ABB RAPID module: Data.modx

MODULE Data
     ! Home
    CONST robtarget rHomePos:=[[368.56,0,469.95],[0.0562068,-0.220361,0.97346,-0.0256232],[0,-1,-1,0],[9E+09,9E+09,9E+09,9E+09,9E+09,9E+09]];

    ! DipSchoko
    CONST robtarget rApprochPickBiscuit:=[[599.81,297.31,218.70],[0.0160586,-0.550955,-0.834314,-0.010557],[0,0,1,0],[9E+09,9E+09,9E+09,9E+09,9E+09,9E+09]];
    CONST robtarget rPickBiscuit:=[[446.88,365.89,48.98],[0.0160535,-0.55171,-0.833815,-0.0105633],[0,0,1,0],[9E+09,9E+09,9E+09,9E+09,9E+09,9E+09]];
    CONST robtarget rPickBiscuitFrame:=[[100,200,300],[1,0,0,0],[0,0,0,0],[9E9,9E9,9E9,9E9,9E9,9E9]];
    CONST robtarget rApprochFontain:=[[610.26,-23.48,232.21],[0.00126836,-0.515151,0.819206,-0.252028],[0,-1,-1,0],[9E+09,9E+09,9E+09,9E+09,9E+09,9E+09]];
    CONST robtarget rDipOnFontainStart:=[[759.86,-193.28,240.92],[0.0169761,-0.705672,0.64261,-0.297977],[-1,-1,-1,0],[9E+09,9E+09,9E+09,9E+09,9E+09,9E+09]];
    CONST robtarget rDipOnFontainEnd:=[[759.85,134.90,240.93],[0.0170012,-0.705702,0.642577,-0.297978],[0,-1,-1,0],[9E+09,9E+09,9E+09,9E+09,9E+09,9E+09]];
    CONST robtarget rApprochVisitor:=[[430.06,-67.55,307.33],[0.0652026,0.183677,-0.814221,0.54686],[0,-1,0,0],[9E+09,9E+09,9E+09,9E+09,9E+09,9E+09]];
    CONST robtarget rGiveVisitor:=[[545.44,-429.78,271.80],[0.078301,0.192469,-0.813094,0.543785],[-1,-2,0,0],[9E+09,9E+09,9E+09,9E+09,9E+09,9E+09]];
    CONST robtarget rPickTowelVisitor:=[[456.74,-234.02,94.25],[1.20556E-05,-0.547416,-0.836861,3.23522E-06],[-1,-1,0,0],[9E+09,9E+09,9E+09,9E+09,9E+09,9E+09]];
    CONST robtarget rGiveTowelToVisitor:=[[471.49,-420.42,179.89],[0.269117,0.480295,0.726977,-0.410361],[-1,-2,1,0],[9E+09,9E+09,9E+09,9E+09,9E+09,9E+09]];
    CONST robtarget rPickBiscuitGripper:=[[456.62,333.14,54.73],[0.584717,-0.596408,0.392302,0.385359],[0,1,-3,0],[9E+09,9E+09,9E+09,9E+09,9E+09,9E+09]];
    CONST robtarget rApprochGiveBiscuitGripper:=[[457.50,-25.27,225.76],[0.00477249,0.835513,-0.549422,-0.00548782],[-1,-1,-2,0],[9E+09,9E+09,9E+09,9E+09,9E+09,9E+09]];
    CONST robtarget rGiveBiscuitGripper:=[[457.53,-410.01,198.66],[0.516342,0.656863,-0.437246,0.332772],[-1,-2,-1,0],[9E+09,9E+09,9E+09,9E+09,9E+09,9E+09]];

    !Demo
    CONST robtarget rDemo_1:=[[337.10,60.43,638.78],[0.179546,0.262059,-0.935203,0.156473],[0,-1,0,0],[9E+09,9E+09,9E+09,9E+09,9E+09,9E+09]];
    CONST robtarget rDemo_2:=[[337.10,60.43,638.78],[0.0792349,0.836164,-0.471453,0.268858],[0,-1,-2,0],[9E+09,9E+09,9E+09,9E+09,9E+09,9E+09]];
    CONST robtarget rDemo_3:=[[387.88,146.46,434.65],[0.203114,0.321731,-0.924772,-0.00560681],[0,0,-1,0],[9E+09,9E+09,9E+09,9E+09,9E+09,9E+09]];
    CONST robtarget rDemo_4:=[[387.88,146.46,434.65],[0.137427,-0.440453,-0.874687,-0.148449],[0,0,0,0],[9E+09,9E+09,9E+09,9E+09,9E+09,9E+09]];
    CONST robtarget rDemo_5:=[[113.57,225.38,350.30],[0.328521,-0.326661,-0.704734,-0.537323],[0,0,0,0],[9E+09,9E+09,9E+09,9E+09,9E+09,9E+09]];
    CONST robtarget rDemo_6:=[[113.57,225.38,350.30],[0.00654879,0.7789,0.627023,0.0107197],[0,-1,1,0],[9E+09,9E+09,9E+09,9E+09,9E+09,9E+09]];
    CONST robtarget rDemo_7:=[[419.91,110.19,470.12],[0.0813147,0.203583,0.920682,-0.322935],[0,-1,0,0],[9E+09,9E+09,9E+09,9E+09,9E+09,9E+09]];
    !TransportPosition
    CONST jointtarget rTransportPosition:=[[0,0,85,0,0,0],[9E9,9E9,9E9,9E9,9E9,9E9]];
ENDMODULE
